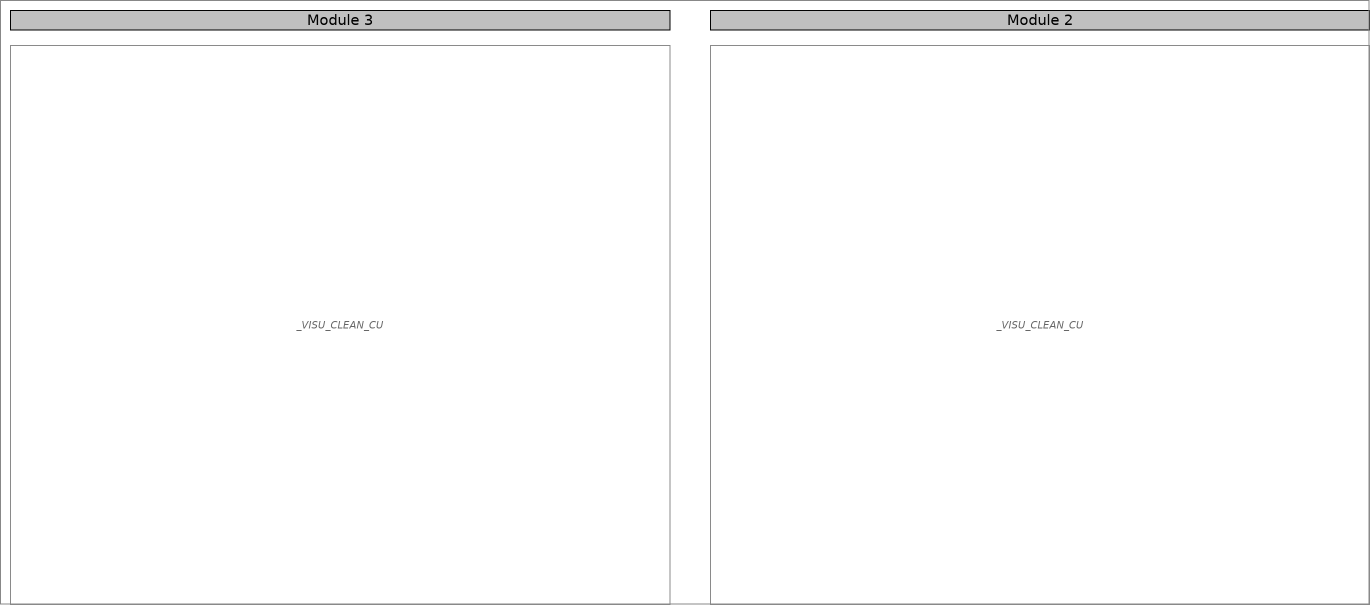
VISUALIZATION VISU_CLEAN_CU  // 1370x605
    Frame (10,45 660x560)
        shows _VISU_CLEAN_CU(m_Inst := 2)
    Rectangle (10,10 660x20), "Module 3"
    Rectangle (710,10 660x20), "Module 2"
    Frame (710,45 660x560)
        shows _VISU_CLEAN_CU(m_Inst := 1)
END_VISUALIZATION

(* stored: Version 1.1.0.1, ProductVersion 3.1.4024.9
   Visu VISU_CLEAN_CU: Id {32b797bd-690e-4d5b-ac84-4ed2747cf92d} *)
